PROGRAM MAIN
VAR
	fbBuilGroup: CfgBuildExt3DGroup;
	fbExecute: FB_Execute;
	fbChannelReset: FB_ChannelReset;

	fbStartStop: FB_ChannelStartStop;
	rtSlideStart:R_TRIG;

	tmrReset: TON;

	fbSelectPrg: FB_SelectProgram;

	fbReleaseGroup: CfgReconfigGroup;

	fbEnable: FB_AxisEnable;
END_VAR

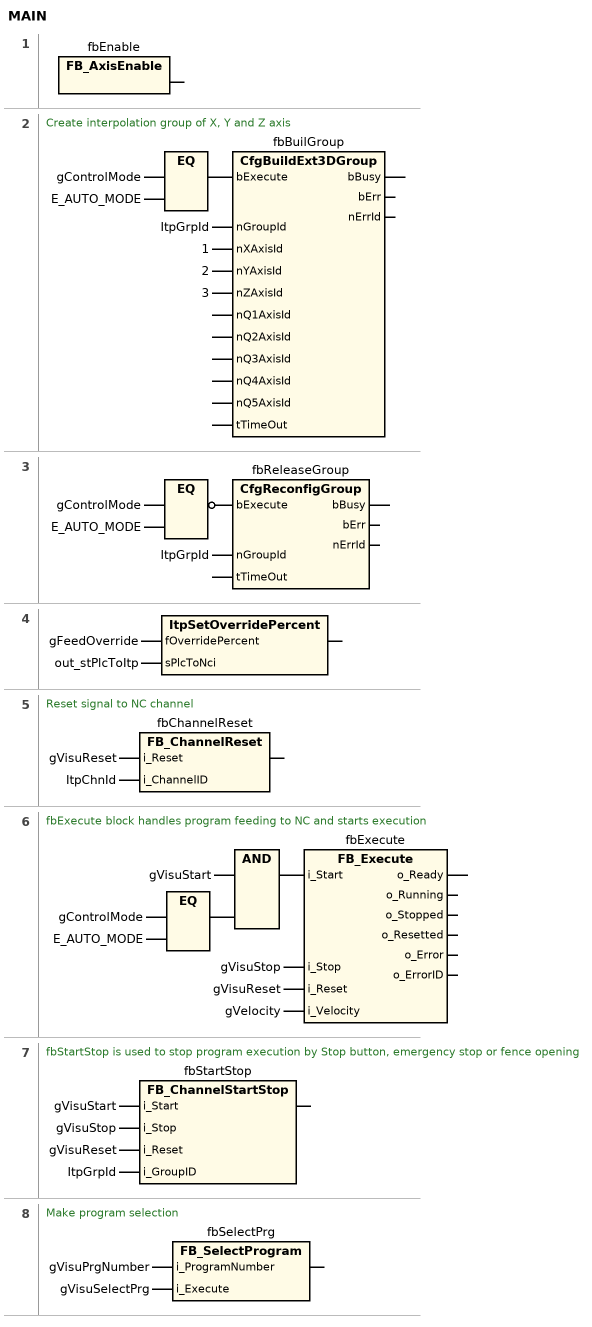
// NETWORK 1
fbEnable(); // FB_AxisEnable

// NETWORK 2
// Create interpolation group of X, Y and Z axis
fbBuilGroup(
    bExecute := gControlMode = E_AUTO_MODE,
    nGroupId := ItpGrpId,
    nXAxisId := 1,
    nYAxisId := 2,
    nZAxisId := 3); // CfgBuildExt3DGroup

// NETWORK 3
fbReleaseGroup(bExecute := NOT (gControlMode = E_AUTO_MODE), nGroupId := ItpGrpId); // CfgReconfigGroup

// NETWORK 4
ItpSetOverridePercent(fOverridePercent := gFeedOverride, sPlcToNci := out_stPlcToItp);

// NETWORK 5
// Reset signal to NC channel
fbChannelReset(i_Reset := gVisuReset, i_ChannelID := ItpChnId); // FB_ChannelReset

// NETWORK 6
// fbExecute block handles program feeding to NC and starts execution
fbExecute(
    i_Start := gVisuStart AND gControlMode = E_AUTO_MODE,
    i_Stop := gVisuStop,
    i_Reset := gVisuReset,
    i_Velocity := gVelocity); // FB_Execute

// NETWORK 7
// fbStartStop is used to stop program execution by Stop button, emergency stop or fence opening
fbStartStop(i_Start := gVisuStart, i_Stop := gVisuStop, i_Reset := gVisuReset, i_GroupID := ItpGrpId); // FB_ChannelStartStop

// NETWORK 8
// Make program selection
fbSelectPrg(i_ProgramNumber := gVisuPrgNumber, i_Execute := gVisuSelectPrg); // FB_SelectProgram

END_PROGRAM

(* stored: Version 1.1.0.1, ProductVersion 3.1.4024.10
   POU MAIN: Id {22c306b9-ad45-460a-b059-bcd54ff7de0f}, SpecialFunc None *)
